TYPE TcoTixonPickVibro_Config_v_1_x_x EXTENDS TcoTixonGenericPickConfig : STRUCT
    {attribute addProperty Name "<#Feeder blow B on start#> - T_FEEDER_BLOWB_ON"}
    FeederBlowBStartTime : TIME := T#300MS;
    {attribute addProperty Name "<#Feeder full blow B time after#> - T_FEEDER_BLOWB_FULL"}
    FeederBlowBFullTime : TIME := T#1S;
    {attribute addProperty Name "<#Feeder blow B  active #>"}
    FeederBlowBActive : BOOL := FALSE;
    {attribute addProperty Name "<#Error time separator #> - T_SEP_ERROR"}
    ErrorTimeSeparator : TIME := T#0S;
    {attribute addProperty Name "<#Error time buffer #> - T_BUFF_ERROR"}
    ErrorTimeBuffer : TIME := T#0S;
    {attribute addProperty Name "<#Error time Hopper #> - T_HOP_ERROR"}
    ErrorTimeHopper : TIME := T#0S;
END_STRUCT
END_TYPE

(* stored: Version 1.1.0.1, ProductVersion 3.1.4024.12
   DUT TcoTixonPickVibro_Config_v_1_x_x: Id {58401dc2-9300-00c2-1af3-6ff07550ac74} *)
